Omron CX-Programmer project 新工程 (CX-Programmer 9.73)

# PLC 新PLC1: CPM2* 

## Global symbols (name address type ; comment)
0 CHANNEL  ; 密码设置
0.00 BOOL  ; 故障复位SB7
0.01 BOOL  ; 飞轮制动SA2-2
0.02 BOOL  ; 强制润滑SA3
0.03 BOOL  ; 脚踏操作SF
0.04 BOOL  ; 手动操作SB8
0.05 BOOL  ; 寸动操作SA5-1
0.06 BOOL  ; 单次操作SA5-2
0.07 BOOL  ; 连续操作SA5-3
0.08 BOOL  ; 主电机运行KM2
0.09 BOOL  ; 主电机过载FR1
0.10 BOOL  ; 润滑电机运行KM4
0.11 BOOL  ; 润滑电机过载FR2
10.00 BOOL  ; 计数器PC
10.02 BOOL  ; 寸动延时继电器
10.03 BOOL  ; 吹件计数器
10.04 BOOL  ; 润滑泵运行KM4
10.05 BOOL  ; 润滑指示灯
10.06 BOOL  ; 卸荷指示灯
10.07 BOOL  ; 二度落灯
10.08 BOOL  ; 离合器接通2
10.09 BOOL  ; 制动器脱开2
11.00 BOOL  ; 气压不足灯HL3
11.01 BOOL  ; 滑块超程灯HL4
11.02 BOOL  ; 压机超载灯HL5
11.03 BOOL  ; 衬套超温灯HL6
11.04 BOOL  ; 压机就绪灯HL7
11.05 BOOL  ; 润滑指示灯HL8
11.06 BOOL  ; 润滑故障灯HL9
11.07 BOOL  ; 飞轮制动灯HL10
12.00 BOOL  ; 吹件阀
12.01 BOOL  ; 制动器脱开
12.02 BOOL  ; 制动器Y1
12.03 BOOL  ; 制动器Y2
12.04 BOOL  ; 离合器Y3
12.05 BOOL  ; 离合器Y4
12.06 BOOL  ; 飞轮制动Y5
12.07 BOOL  ; 卸荷阀
12.13 BOOL  ; 吹件计数阀动作准
13.00 BOOL  ; 吨位故障
13.01 BOOL  ; 温度故障
13.02 BOOL  ; 润滑故障发现点
13.03 BOOL  ; 润滑故障确认点
13.04 BOOL  ; 气压异常故障
13.05 BOOL  ; 分油器故障
14.00 BOOL  ; 准备运行
14.01 BOOL  ; 锻压
14.02 BOOL  ; 锻压停车
14.03 BOOL  ; 正常结束
15.00 BOOL  ; 压机超载1报警
15.01 BOOL  ; 压机超载2报警
15.02 BOOL  ; 油路异常
15.03 BOOL  ; 温度超温故障
15.04 BOOL  ; 润滑故障点
15.05 BOOL  ; 润滑故障确认
15.10 BOOL  ; 干油泵超载中继
15.11 BOOL  ; 润滑电机过载
16.00 BOOL  ; 一次真正故障
16.03 BOOL  ; 制动器脱开1
16.04 BOOL  ; 离合器接通1
16.05 BOOL  ; 制动器脱开2
16.06 BOOL  ; 离合器接通2
16.07 BOOL  ; 润滑保持
16.08 BOOL  ; 润滑1故障
16.09 BOOL  ; 润滑2故障
16.10 BOOL  ; 检测保持
16.14 BOOL  ; 脚踏延时接通
17.00 BOOL  ; 连打
1.00 BOOL  ; 压机超载1KA2
1.01 BOOL  ; 压机超载2KA3
1.02 BOOL  ; 吨位超负荷
1.03 BOOL  ; 气压检测SP1
1.04 BOOL  ; 左右杆衬套超温
1.05 BOOL  ; 干油泵超载SP2
1.06 BOOL  ; 干油脂低位SQ9
1.07 BOOL  ; 分油器动作
1.08 BOOL  ; 分油器二堵塞
1.09 BOOL  ; 分油器三堵塞
1.10 BOOL  ; 分油器四堵塞
1.11 BOOL  ; 油脂低位2
2 CHANNEL  ; 延时离合
2.00 BOOL  ; 油脂堵塞2
2.01 BOOL  ; 润滑监控2
2.02 BOOL  ; 气压正常
2.03 BOOL  ; 手动润滑
2.04 BOOL  ; 上死点
2.05 BOOL  ; 滑块上位B11
2.06 BOOL  ; 滑块运行B12
2.07 BOOL  ; 离合器断开一B13
2.08 BOOL  ; 制动器脱开一B14
2.09 BOOL  ; 离合器断开二B15
2.10 BOOL  ; 制动器脱开二B16
2.11 BOOL  ; 滑块超程凸轮
AR10.01 BOOL  ; 加密指令
TIM001 BOOL  ; 润滑故障点延时
TIM002 BOOL  ; 连续操作延时
TIM003 BOOL  ; 脚踏延时
TIM004 BOOL  ; 润滑时间
TIM005 BOOL  ; 打击次数到延时
TIM006 BOOL  ; 延时开通
TIM007 BOOL  ; 延时接通
TIM008 BOOL  ; 延时完成比较
TIM010 BOOL  ; 延时制动
TIM011 BOOL  ; 润滑阀动作时间
TIM011 BOOL  ; 润滑阀循环打油次
TIM011 BOOL  ; 一次润滑结束
TIM012 BOOL  ; 润滑阀动作时间
TIM013 BOOL  ; 延时开通
TIM014 BOOL  ; 延时接通
TIM020 BOOL  ; 润滑确定计数
TIM020 BOOL  ; 润滑故障次数
TIM021 BOOL  ; 故障标记
TIM021 BOOL  ; 故障
TIM022 BOOL  ; 连续操作
TIM023 BOOL  ; 滑块动作次数
TIM023 BOOL  ; 滑块打击次数
TIM024 BOOL  ; 电机每次启动标志
TIM025 BOOL  ; 行程计数
TIM025 BOOL  ; 行程计数
TIM026 BOOL  ; 开机已润滑过标志
TIM027 BOOL  ; 分油器计数
TIM028 BOOL  ; 一次润滑故障
TIM029 BOOL  ; 分油器多次故障
TIM030 BOOL  ; 分油器动作次数
TIM031 BOOL  ; 标志为ON接通
TIM031 BOOL  ; 故障计数
TIM033 BOOL  ; 标志为ON接通
TIM034 BOOL  ; 延时恢复初始状态
TIM045 BOOL  ; 延时断开

## Program 新程序1 (no task)
; 这个项目实现了一个1600吨压力机的控制系统，包含压力机启停、锻压动作、润滑系统及故障监测模块，用于控制重型锻压设备。系统支持手动、寸动、单次和连续等多种操作模式（互斥），通过操作面板按钮和传感器信号实现压力机的运行管理。 / 设备：压力机、润滑系统、离合器、制动器、传感器和操作面板。 / 系统通过操作面板按钮如故障复位和脚踏操作采集输入信号。传感器信号如气压检测和干油泵超载用于监测设备状态。 / 当脚踏操作按下时，只有在准备运行置位且滑块在上位时，锻压动作才会启动。锻压动作启动前，润滑故障为假时才允许运行，以确保润滑系统正常。锻压动作置位时，触发离合器接通和制动器脱开的准备。 / 润滑时间用于控制润滑泵的运行周期。润滑泵运行由润滑保持触发。润滑系统由润滑时间控制周期，到时后润滑泵运行停止。系统启动前，滑块在上位且无故障时，置位准备运行。准备运行置位后，点亮压机就绪灯。 / 气压不足触发时，点亮气压不足灯。气压不足触发时，暂停锻压动作。干油泵超载或润滑电机过载触发时，点亮润滑故障灯。干油泵超载或润滑电机过载触发时，停止润滑。润滑故障灯在润滑故障如润滑故障计数器触发时点亮。 / 故障复位按下后，重置故障状态如计数器和润滑故障。制动动作由延时制动计时1个单位时间后触发。压机超载1报警由传感器触发，超载2报警由另一传感器触发。离合器接通由锻压状态和寸动操作控制。制动器脱开由锻压状态和寸动操作控制。 / 打击次数达到10次后触发润滑保持的计时。润滑保持由计时启动。分油器动作配合计时和计数器监测润滑状态。润滑故障计数器用于记录分油器动作的异常次数。连续操作由计数器触发，并在延时40个单位时间后准备。 / 锻压停车在制动器和离合器状态正确时置位。正常结束在滑块上位且锻压停车置位时触发。飞轮制动控制Y5输出。Y5输出置位时点亮飞轮制动灯。

### Section 段1

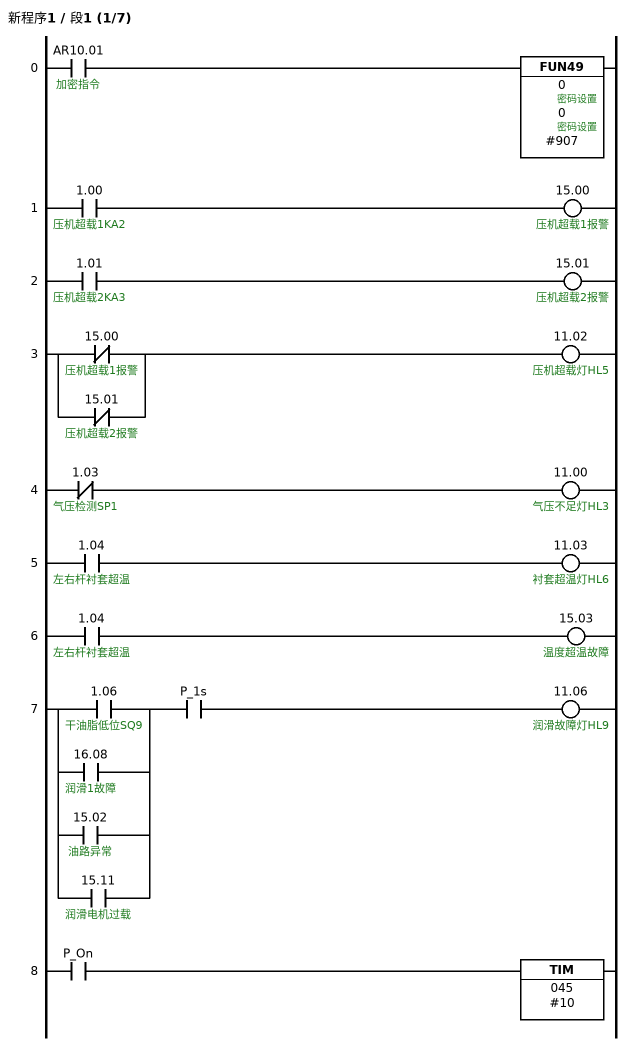
; rung 0
LD AR10.01  ; 加密指令
FUN49 0 0 #907  ; 密码设置
; rung 1
LD 1.00  ; 压机超载1KA2
OUT 15.00  ; 压机超载1报警
; rung 2
LD 1.01  ; 压机超载2KA3
OUT 15.01  ; 压机超载2报警
; rung 3
LDNOT 15.00  ; 压机超载1报警
ORNOT 15.01  ; 压机超载2报警
OUT 11.02  ; 压机超载灯HL5
; rung 4
LDNOT 1.03  ; 气压检测SP1
OUT 11.00  ; 气压不足灯HL3
; rung 5
LD 1.04  ; 左右杆衬套超温
OUT 11.03  ; 衬套超温灯HL6
; rung 6
LD 1.04  ; 左右杆衬套超温
OUT 15.03  ; 温度超温故障
; rung 7
LD 1.06  ; 干油脂低位SQ9
OR 16.08  ; 润滑1故障
OR 15.02  ; 油路异常
OR 15.11  ; 润滑电机过载
AND P_1s
OUT 11.06  ; 润滑故障灯HL9
; rung 8
LD P_On
TIM 045 #10

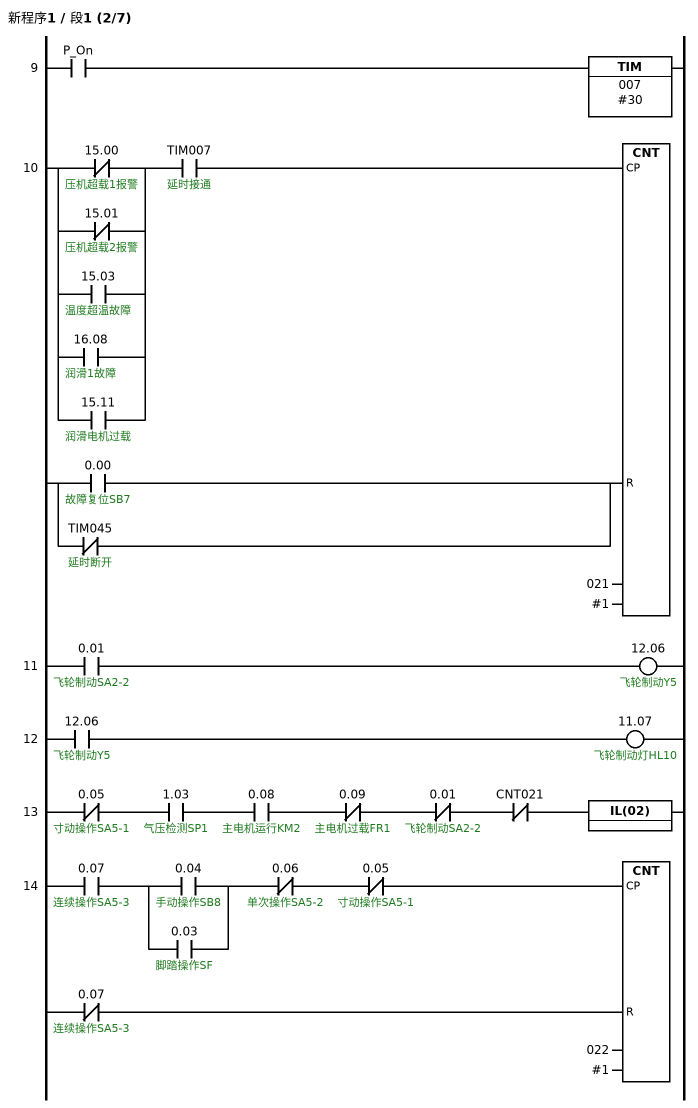
; rung 9
LD P_On
TIM 007 #30
; rung 10
LDNOT 15.00  ; 压机超载1报警
ORNOT 15.01  ; 压机超载2报警
OR 15.03  ; 温度超温故障
OR 16.08  ; 润滑1故障
OR 15.11  ; 润滑电机过载
AND TIM007  ; 延时接通
LD 0.00  ; 故障复位SB7
ORNOT TIM045  ; 延时断开
CNT 021 #1
; rung 11
LD 0.01  ; 飞轮制动SA2-2
OUT 12.06  ; 飞轮制动Y5
; rung 12
LD 12.06  ; 飞轮制动Y5
OUT 11.07  ; 飞轮制动灯HL10
; rung 13
LDNOT 0.05  ; 寸动操作SA5-1
AND 1.03  ; 气压检测SP1
AND 0.08  ; 主电机运行KM2
ANDNOT 0.09  ; 主电机过载FR1
ANDNOT 0.01  ; 飞轮制动SA2-2
ANDNOT CNT021
IL(02)
; rung 14
LD 0.07  ; 连续操作SA5-3
LD 0.04  ; 手动操作SB8
OR 0.03  ; 脚踏操作SF
ANDLD
ANDNOT 0.06  ; 单次操作SA5-2
ANDNOT 0.05  ; 寸动操作SA5-1
LDNOT 0.07  ; 连续操作SA5-3
CNT 022 #1

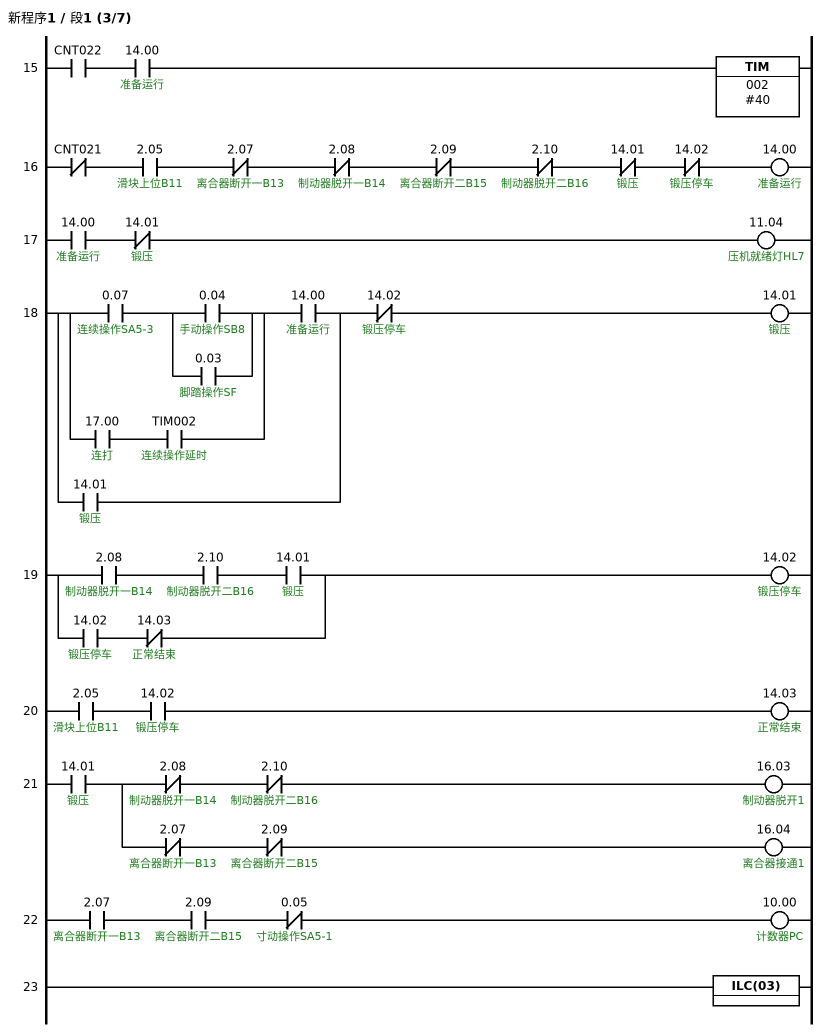
; rung 15
LD CNT022
AND 14.00  ; 准备运行
TIM 002 #40
; rung 16
LDNOT CNT021
AND 2.05  ; 滑块上位B11
ANDNOT 2.07  ; 离合器断开一B13
ANDNOT 2.08  ; 制动器脱开一B14
ANDNOT 2.09  ; 离合器断开二B15
ANDNOT 2.10  ; 制动器脱开二B16
ANDNOT 14.01  ; 锻压
ANDNOT 14.02  ; 锻压停车
OUT 14.00  ; 准备运行
; rung 17
LD 14.00  ; 准备运行
ANDNOT 14.01  ; 锻压
OUT 11.04  ; 压机就绪灯HL7
; rung 18
LD 0.07  ; 连续操作SA5-3
LD 0.04  ; 手动操作SB8
OR 0.03  ; 脚踏操作SF
ANDLD
LD 17.00  ; 连打
AND TIM002  ; 连续操作延时
ORLD
AND 14.00  ; 准备运行
OR 14.01  ; 锻压
ANDNOT 14.02  ; 锻压停车
OUT 14.01  ; 锻压
; rung 19
LD 2.08  ; 制动器脱开一B14
AND 2.10  ; 制动器脱开二B16
AND 14.01  ; 锻压
LD 14.02  ; 锻压停车
ANDNOT 14.03  ; 正常结束
ORLD
OUT 14.02  ; 锻压停车
; rung 20
LD 2.05  ; 滑块上位B11
AND 14.02  ; 锻压停车
OUT 14.03  ; 正常结束
; rung 21
LD 14.01  ; 锻压
OUT TR0
ANDNOT 2.08  ; 制动器脱开一B14
ANDNOT 2.10  ; 制动器脱开二B16
OUT 16.03  ; 制动器脱开1
LD TR0
ANDNOT 2.07  ; 离合器断开一B13
ANDNOT 2.09  ; 离合器断开二B15
OUT 16.04  ; 离合器接通1
; rung 22
LD 2.07  ; 离合器断开一B13
AND 2.09  ; 离合器断开二B15
ANDNOT 0.05  ; 寸动操作SA5-1
OUT 10.00  ; 计数器PC
; rung 23
ILC(03)

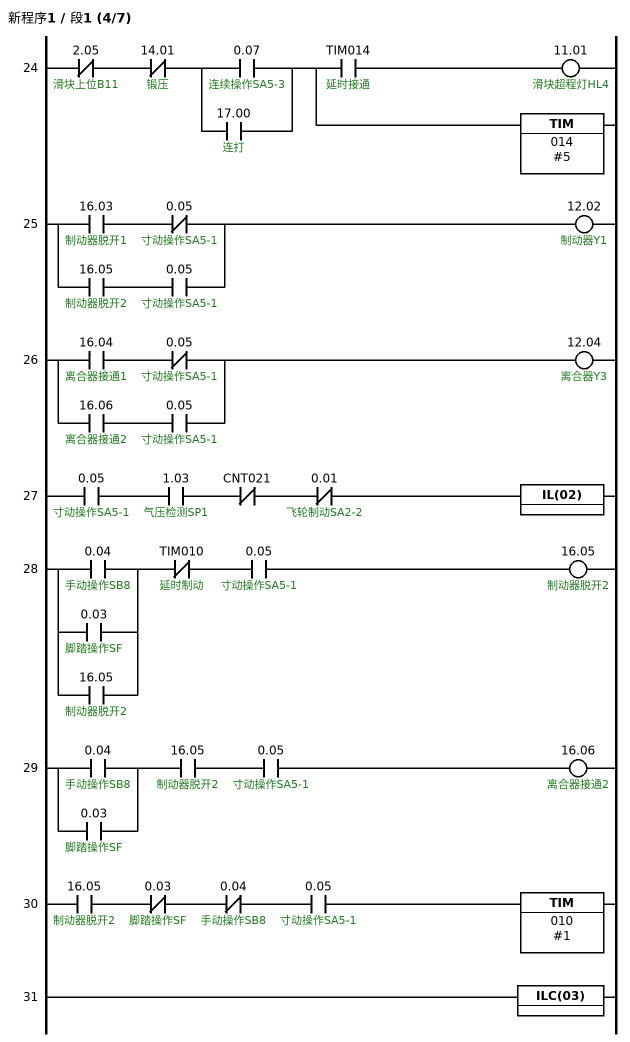
; rung 24
LDNOT 2.05  ; 滑块上位B11
ANDNOT 14.01  ; 锻压
LD 0.07  ; 连续操作SA5-3
OR 17.00  ; 连打
ANDLD
OUT TR0
AND TIM014  ; 延时接通
OUT 11.01  ; 滑块超程灯HL4
LD TR0
TIM 014 #5
; rung 25
LD 16.03  ; 制动器脱开1
ANDNOT 0.05  ; 寸动操作SA5-1
LD 16.05  ; 制动器脱开2
AND 0.05  ; 寸动操作SA5-1
ORLD
OUT 12.02  ; 制动器Y1
; rung 26
LD 16.04  ; 离合器接通1
ANDNOT 0.05  ; 寸动操作SA5-1
LD 16.06  ; 离合器接通2
AND 0.05  ; 寸动操作SA5-1
ORLD
OUT 12.04  ; 离合器Y3
; rung 27
LD 0.05  ; 寸动操作SA5-1
AND 1.03  ; 气压检测SP1
ANDNOT CNT021
ANDNOT 0.01  ; 飞轮制动SA2-2
IL(02)
; rung 28
LD 0.04  ; 手动操作SB8
OR 0.03  ; 脚踏操作SF
OR 16.05  ; 制动器脱开2
ANDNOT TIM010  ; 延时制动
AND 0.05  ; 寸动操作SA5-1
OUT 16.05  ; 制动器脱开2
; rung 29
LD 0.04  ; 手动操作SB8
OR 0.03  ; 脚踏操作SF
AND 16.05  ; 制动器脱开2
AND 0.05  ; 寸动操作SA5-1
OUT 16.06  ; 离合器接通2
; rung 30
LD 16.05  ; 制动器脱开2
ANDNOT 0.03  ; 脚踏操作SF
ANDNOT 0.04  ; 手动操作SB8
AND 0.05  ; 寸动操作SA5-1
TIM 010 #1
; rung 31
ILC(03)

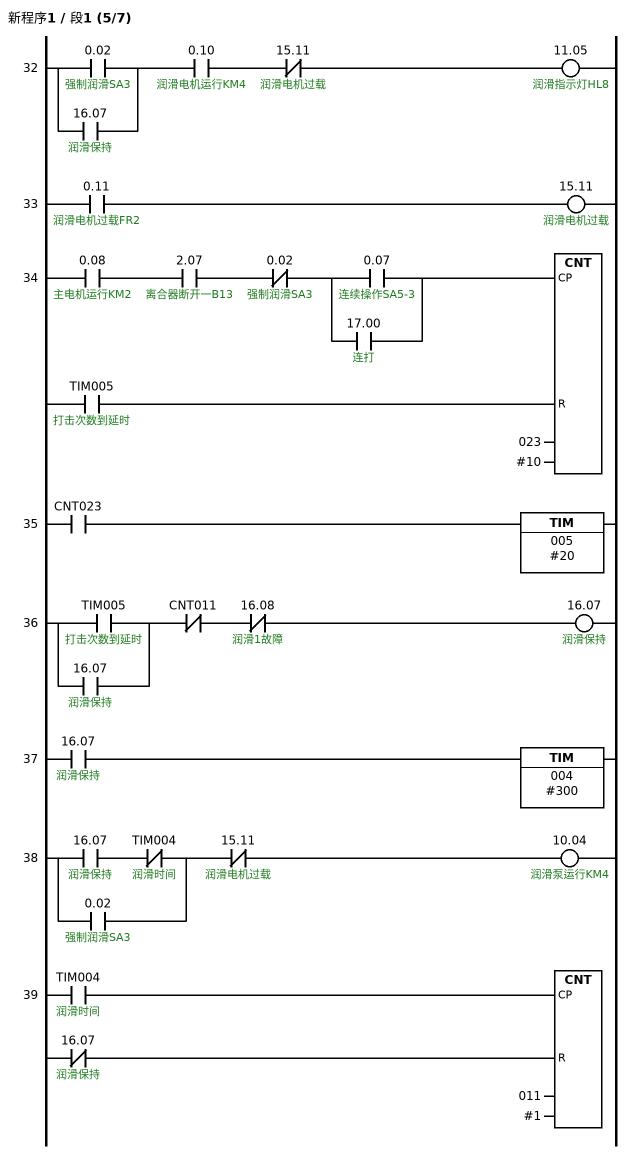
; rung 32
LD 0.02  ; 强制润滑SA3
OR 16.07  ; 润滑保持
AND 0.10  ; 润滑电机运行KM4
ANDNOT 15.11  ; 润滑电机过载
OUT 11.05  ; 润滑指示灯HL8
; rung 33
LD 0.11  ; 润滑电机过载FR2
OUT 15.11  ; 润滑电机过载
; rung 34
LD 0.08  ; 主电机运行KM2
AND 2.07  ; 离合器断开一B13
ANDNOT 0.02  ; 强制润滑SA3
LD 0.07  ; 连续操作SA5-3
OR 17.00  ; 连打
ANDLD
LD TIM005  ; 打击次数到延时
CNT 023 #10
; rung 35
LD CNT023
TIM 005 #20
; rung 36
LD TIM005  ; 打击次数到延时
OR 16.07  ; 润滑保持
ANDNOT CNT011
ANDNOT 16.08  ; 润滑1故障
OUT 16.07  ; 润滑保持
; rung 37
LD 16.07  ; 润滑保持
TIM 004 #300
; rung 38
LD 16.07  ; 润滑保持
ANDNOT TIM004  ; 润滑时间
OR 0.02  ; 强制润滑SA3
ANDNOT 15.11  ; 润滑电机过载
OUT 10.04  ; 润滑泵运行KM4
; rung 39
LD TIM004  ; 润滑时间
LDNOT 16.07  ; 润滑保持
CNT 011 #1

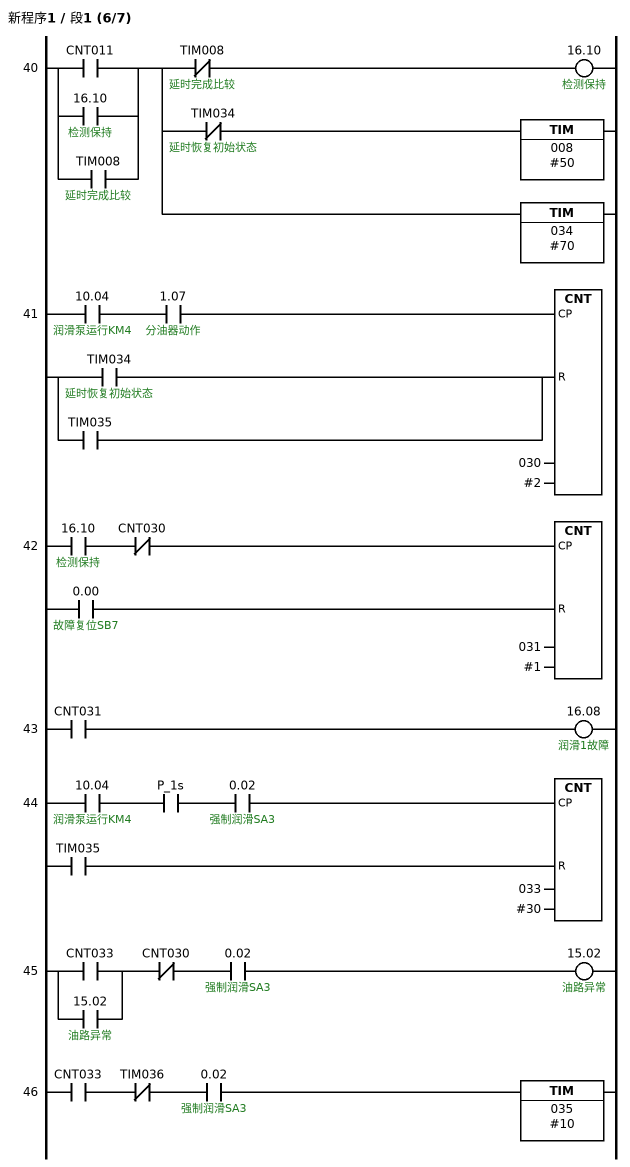
; rung 40
LD CNT011
OR 16.10  ; 检测保持
OR TIM008  ; 延时完成比较
OUT TR0
ANDNOT TIM008  ; 延时完成比较
OUT 16.10  ; 检测保持
LD TR0
ANDNOT TIM034  ; 延时恢复初始状态
TIM 008 #50
LD TR0
TIM 034 #70
; rung 41
LD 10.04  ; 润滑泵运行KM4
AND 1.07  ; 分油器动作
LD TIM034  ; 延时恢复初始状态
OR TIM035
CNT 030 #2
; rung 42
LD 16.10  ; 检测保持
ANDNOT CNT030
LD 0.00  ; 故障复位SB7
CNT 031 #1
; rung 43
LD CNT031
OUT 16.08  ; 润滑1故障
; rung 44
LD 10.04  ; 润滑泵运行KM4
AND P_1s
AND 0.02  ; 强制润滑SA3
LD TIM035
CNT 033 #30
; rung 45
LD CNT033
OR 15.02  ; 油路异常
ANDNOT CNT030
AND 0.02  ; 强制润滑SA3
OUT 15.02  ; 油路异常
; rung 46
LD CNT033
ANDNOT TIM036
AND 0.02  ; 强制润滑SA3
TIM 035 #10

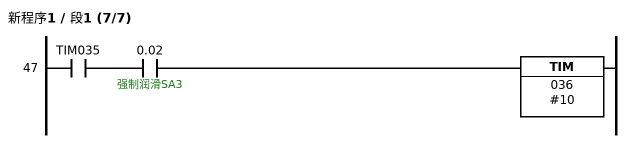
; rung 47
LD TIM035
AND 0.02  ; 强制润滑SA3
TIM 036 #10
; rung 48
END(01)